TYPE NightReduction :
STRUCT
	EN: BOOL;
	StartTime: DT;
	StopTime: DT;
	SupplyAirFan: LREAL;
	ExtractAitFan: LREAL;
END_STRUCT
END_TYPE

(* stored: Version 1.1.0.1, ProductVersion 3.1.4024.6
   DUT NightReduction: Id {29c0e371-e0b5-4f01-854c-edf6a97a8314} *)
